// TIA Portal V19 export
TYPE "Straightener_Status"
   STRUCT
      Feed : "PositioningMachine_COut";
      Lift_Entry : "ValveMachine_COut";
      Lift_Exit : "ValveMachine_COut";
   END_STRUCT;
END_TYPE
